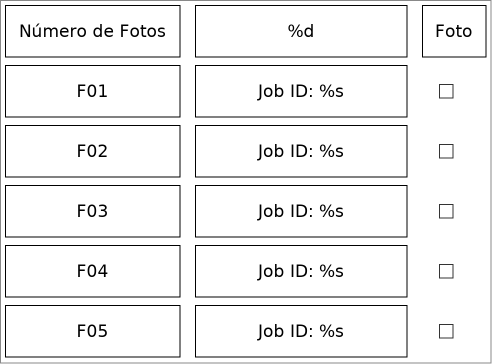
VISUALIZATION Lista_PontosRoboCamera  // 492x364
    Rectangle (5,5 175x52), "Número de Fotos"
    Rectangle (195,5 212x52), "%d", text variable: Recipe_Pontos_Camera_Select, input disabled if: Not b_editar_receita and Not b_criar_receita
        OnMouseClick: write the text variable via Default, min 0, max 5
    Rectangle (5,65 175x52), "F01", invisible if: Recipe_Pontos_Camera_Select<1
    Rectangle (195,65 212x52), "Job ID: %s", text variable: Recipe_JobID_F01_Camera_Select, invisible if: Recipe_Pontos_Camera_Select<1, input disabled if: Not b_editar_receita and Not b_criar_receita
        OnMouseClick: write the text variable via Default, min 0, max 500
    Rectangle (5,125 175x52), "F02", invisible if: Recipe_Pontos_Camera_Select<2
    Rectangle (195,125 212x52), "Job ID: %s", text variable: Recipe_JobID_F02_Camera_Select, invisible if: Recipe_Pontos_Camera_Select<2, input disabled if: Not b_editar_receita and Not b_criar_receita
        OnMouseClick: write the text variable via Default, min 0, max 500
    Rectangle (5,185 175x52), "F03", invisible if: Recipe_Pontos_Camera_Select<3
    Rectangle (195,185 212x52), "Job ID: %s", text variable: Recipe_JobID_F03_Camera_Select, invisible if: Recipe_Pontos_Camera_Select<3, input disabled if: Not b_editar_receita and Not b_criar_receita
        OnMouseClick: write the text variable via Default
    Rectangle (5,245 175x52), "F04", invisible if: Recipe_Pontos_Camera_Select<4
    Rectangle (195,245 212x52), "Job ID: %s", text variable: Recipe_JobID_F04_Camera_Select, invisible if: Recipe_Pontos_Camera_Select<4, input disabled if: Not b_editar_receita and Not b_criar_receita
        OnMouseClick: write the text variable via Default
    Rectangle (5,305 175x52), "F05", invisible if: Recipe_Pontos_Camera_Select<5
    Rectangle (195,305 212x52), "Job ID: %s", text variable: Recipe_JobID_F05_Camera_Select, invisible if: Recipe_Pontos_Camera_Select<5, input disabled if: Not b_editar_receita and Not b_criar_receita
        OnMouseClick: write the text variable via Default
    Rectangle (422,5 64x52), "Foto"
    Checkbox (437,71 40x40), variable: TRUE, invisible if: Recipe_Pontos_Camera_Select<1, input disabled if: TRUE
    Checkbox (437,131 40x40), variable: TRUE, invisible if: Recipe_Pontos_Camera_Select<2, input disabled if: TRUE
    Checkbox (437,191 40x40), variable: TRUE, invisible if: Recipe_Pontos_Camera_Select<3, input disabled if: TRUE
    Checkbox (437,251 40x40), variable: TRUE, invisible if: Recipe_Pontos_Camera_Select<4, input disabled if: TRUE
    Checkbox (437,311 40x40), variable: TRUE, invisible if: Recipe_Pontos_Camera_Select<5, input disabled if: TRUE
END_VISUALIZATION

(* stored: Version 1.1.0.1, ProductVersion 3.1.4024.11
   Visu Lista_PontosRoboCamera: Id {e6d60e9b-10a4-489e-b2a5-4455a9f2d807} *)
